PROGRAM MAIN
VAR
END_VAR

P_EnOCean();

END_PROGRAM

(* stored: Version 1.1.0.1, ProductVersion 3.1.4024.0
   POU MAIN: Id {6bc8b873-5d1d-44dc-88d5-c781d1258060}, SpecialFunc None *)
